//设备报警信息打印
FUNCTION error_Printf : BOOL
VAR_INPUT
	errorID					:DINT;
END_VAR
VAR
	sErrTXT					:STRING(255);
	sErrWTXT				:WSTRING(255);
END_VAR

sErrTXT:=errorMonitor.getErrTXT(errorID);
sErrWTXT:=errorMonitor.getErrWTXT(errorID);
IF gCNErrShow THEN
	gLog.append_EX(sErrWTXT);
	gErrWTxtShow:=sErrWTXT;
ELSE
	gLog.append(sErrTXT);
	gErrTxtShow:=sErrTXT;
	gErrWTxtShow:=TO_WSTRING(gErrTxtShow);
END_IF

END_FUNCTION

(* stored: Version 1.1.0.1, ProductVersion 3.1.4024.4
   POU error_Printf: Id {e86b548f-0fd1-4186-b6e0-397fbeb0a7dc}, SpecialFunc None *)
